// TIA Portal V20 export
TYPE "UDT_MaintenanceElement"
   STRUCT
      RunTime : Real;   // Temps de fonctionnement actuel (en unité de temps)
      RunTimeSec : Real;   // Temps de fonctionnement actuel (en secondes)
      WarningThreshold : Int;   // Seuil d'avertissement en % (par défaut 80%)
      AlarmThreshold : Int;   // Durée maximale avant maintenance
      TimeUnit : Int;   // Unité de temps (0:Minutes, 1:Hours, 2:Days)
      ResetRunTime : Bool;   // Reset Temps de fonctionnement actuel
   END_STRUCT;
END_TYPE
